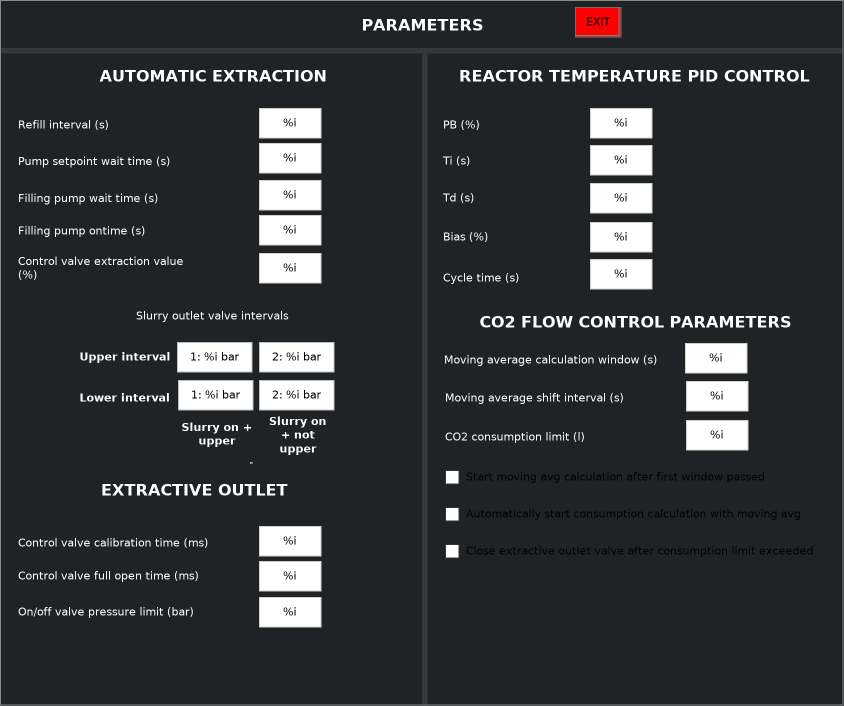
VISUALIZATION ParameterView  // 844x706
    Textfield (259,108 62x30), "%i", text variable: ParameterViewBindings.refillIntervalTextField_TextVariable
        OnMouseDown: write the text variable via VisuDialogs.Numpad, min 1, max 999
    Label (15,103 190x44), "Refill interval (s)"
    Button (575,7 46x30), "EXIT", pressed state: NOT ProcessViewBindings.autoExtractionParameterMenuButton_ToggleVariable
        toggle ProcessViewBindings.autoExtractionParameterMenuButton_ToggleVariable
    Label (15,209 190x44), "Filling pump ontime (s)"
    Label (15,246 190x44), "Control valve extraction value (%)"
    Textfield (259,215 62x30), "%i", text variable: ParameterViewBindings.pumpOnTimeTextField_TextVariable
        OnMouseDown: write the text variable via VisuDialogs.Numpad, min 1, max 5999
    Textfield (259,253 62x30), "%i", text variable: ParameterViewBindings.controlValveOpeningValueTextField_TextVariable
        OnMouseDown: write the text variable via VisuDialogs.Numpad, min 1, max 5999
    Label (15,139 190x45), "Pump setpoint wait time (s)"
    Textfield (259,143 62x30), "%i", text variable: ParameterViewBindings.pumpSetpointWaitTimeTextField_TextVariable
        OnMouseDown: write the text variable via VisuDialogs.Numpad, min 0, max 999
    Image (250,462 2x1), image: VisuSymbols.Symbols.ArrowBoldRight
    Label (75,335 100x44), "Upper interval"
    Label (75,376 100x44), "Lower interval"
    Textfield (177,342 75x30), "1: %i bar", text variable: ParameterViewBindings.UpperIntervalSlurryOnUpperTextField_TextVariable
        OnMouseDown: write the text variable via VisuDialogs.Numpad, min -100, max 100
    Textfield (259,342 75x30), "2: %i bar", text variable: ParameterViewBindings.UpperIntervalSlurryOnNotUpperTextField_TextVariable
        OnMouseDown: write the text variable via VisuDialogs.Numpad, min -100, max 100
    Textfield (178,380 75x30), "1: %i bar", text variable: ParameterViewBindings.LowerIntervalSlurryOnUpperTextField_TextVariable
        OnMouseDown: write the text variable via VisuDialogs.Numpad, min -100, max 100
    Textfield (259,380 75x30), "2: %i bar", text variable: ParameterViewBindings.LowerIntervalSlurryOnNotUpperTextField_TextVariable
        OnMouseDown: write the text variable via VisuDialogs.Numpad, min -100, max 100
    Label (178,412 78x44), "Slurry on + upper"
    Label (262,413 72x44), "Slurry on + not upper"
    Label (5,294 415x44), "Slurry outlet valve intervals"
    Textfield (590,108 62x30), "%i", text variable: ParameterViewBindings.PbTextField_TextVariable
        OnMouseDown: write the text variable via VisuDialogs.Numpad, min 1, max 999
    Label (440,103 103x44), "PB (%)"
    Label (440,139 103x44), "Ti (s)"
    Label (440,176 103x44), "Td (s)"
    Textfield (590,145 62x30), "%i", text variable: ParameterViewBindings.TiTextField_TextVariable
        OnMouseDown: write the text variable via VisuDialogs.Numpad, min 1, max 5999
    Textfield (590,183 62x30), "%i", text variable: ParameterViewBindings.TdTextField_TextVariable
        OnMouseDown: write the text variable via VisuDialogs.Numpad, min 1, max 5999
    Label (440,215 103x44), "Bias (%)"
    Textfield (590,222 62x30), "%i", text variable: ParameterViewBindings.BiasTextField_TextVariable
        OnMouseDown: write the text variable via VisuDialogs.Numpad, min 0, max 999
    Textfield (590,259 62x30), "%i", text variable: ParameterViewBindings.IterationTimeTextField_TextVariable
        OnMouseDown: write the text variable via VisuDialogs.Numpad, min 1, max 5999
    Textfield (259,526 62x30), "%i", text variable: ParameterViewBindings.calibrationTimeTextField_TextVariable
        OnMouseDown: write the text variable via VisuDialogs.Numpad, min 1, max 999999
    Label (15,521 231x44), "Control valve calibration time (ms)"
    Textfield (259,561 62x30), "%i", text variable: ParameterViewBindings.fullOpenTimeTextField_TextVariable
        OnMouseDown: write the text variable via VisuDialogs.Numpad, min 0, max 999999
    Label (15,554 210x44), "Control valve full open time (ms)"
    Label (4,61 419x30), "AUTOMATIC EXTRACTION"
    Label (34,475 321x30), "EXTRACTIVE OUTLET"
    Rectangle (422,50 5x655)
    Label (430,61 409x30), "REACTOR TEMPERATURE PID CONTROL"
    Label (264,10 317x30), "PARAMETERS"
    Label (440,256 117x44), "Cycle time (s)"
    Rectangle (1,48 842x5)
    Label (15,176 190x45), "Filling pump wait time (s)"
    Textfield (259,180 62x30), "%i", text variable: ParameterViewBindings.refillPumpWaitTimeTextField_TextVariable
        OnMouseDown: write the text variable via VisuDialogs.Numpad, min 0, max 999
    Textfield (259,597 62x30), "%i", text variable: ParameterViewBindings.onOffValvePressureLimitTextField_TextVariable
        OnMouseDown: write the text variable via VisuDialogs.Numpad, min 0, max 5999
    Label (15,590 200x44), "On/off valve pressure limit (bar)"
    Label (431,307 409x30), "CO2 FLOW CONTROL PARAMETERS"
    Label (441,338 235x44), "Moving average calculation window (s)"
    Textfield (685,343 62x30), "%i", text variable: ParameterViewBindings.movingAvgWindowTextField_TextVariable
        OnMouseDown: write the text variable via VisuDialogs.Numpad, min 1, max 999
    Label (442,415 235x44), "CO2 consumption limit (l)"
    Textfield (686,420 62x30), "%i", text variable: ParameterViewBindings.co2ConsumptionLimitTextField_TextVariable
        OnMouseDown: write the text variable via VisuDialogs.Numpad, min 0, max 9999
    Label (442,376 235x44), "Moving average shift interval (s)"
    Textfield (686,381 62x30), "%i", text variable: ParameterViewBindings.movingAvgShiftIntervalTextField_TextVariable
        OnMouseDown: write the text variable via VisuDialogs.Numpad, min 0, max 999
    Checkbox (443,462 389x30), "Start moving avg calculation after first window passed", variable: ParameterViewBindings.startMovingAvgAfterWindowCheckBox_Variable
    Checkbox (443,499 388x30), "Automatically start consumption calculation with moving avg", variable: ParameterViewBindings.automaticallyStartConsumptionCalculationCheckBox_variable
    Checkbox (443,536 388x30), "Close extractive outlet valve after consumption limit exceeded", variable: ParameterViewBindings.startMovingAvgAfterWindowCheckBox_Variable
END_VISUALIZATION

(* stored: Version 1.1.0.1, ProductVersion 3.1.4024.9
   Visu ParameterView: Id {800908a7-96e7-46b1-b2c8-3866ec22bff5} *)
